(* PLC project prj, KAIST_DSLAB noNameNow 1, author bwkim *)
(* stored: creationDateTime 2015-7-21T04:57:08, modificationDateTime 2015-7-21T04:57:08 *)

PROGRAM program5____sub1
  VAR
    VF_TON : null;
  END_VAR
  VAR
    VF_PTON : null;
  END_VAR
  VAR_INPUT CONSTANT
    K_DELAY : null;
  END_VAR
  VAR_OUTPUT
    TON_et : null;
  END_VAR
  VAR_OUTPUT
    PTON_et : null;
  END_VAR
  VAR_IN_OUT
    PTRIP_LOGIC : BOOL := FALSE;
  END_VAR
  VAR_IN_OUT
    TRIP_LOGIC : BOOL := FALSE;
  END_VAR
  VAR  (* added by the conversion: wires and edge detectors of the diagram *)
    _SUB_REAL34_OUT : ANY;
    _DIV_REAL56_OUT : INT;
    _SEL_REAL72_OUT : INT;
    _SEL_REAL73_OUT : INT;
    _SEL_REAL74_OUT : INT;
    _SEL_BOOL75_OUT : BOOL;
    _SEL_REAL39_OUT : INT;
    _SEL_BOOL82_OUT : BOOL;
    _SEL_REAL83_OUT : INT;
    _AND2_BOOL63_OUT : BOOL;
    _SEL_REAL86_OUT : INT;
    _SEL_REAL87_OUT : INT;
    _AND2_BOOL41_OUT : ANY;
  END_VAR

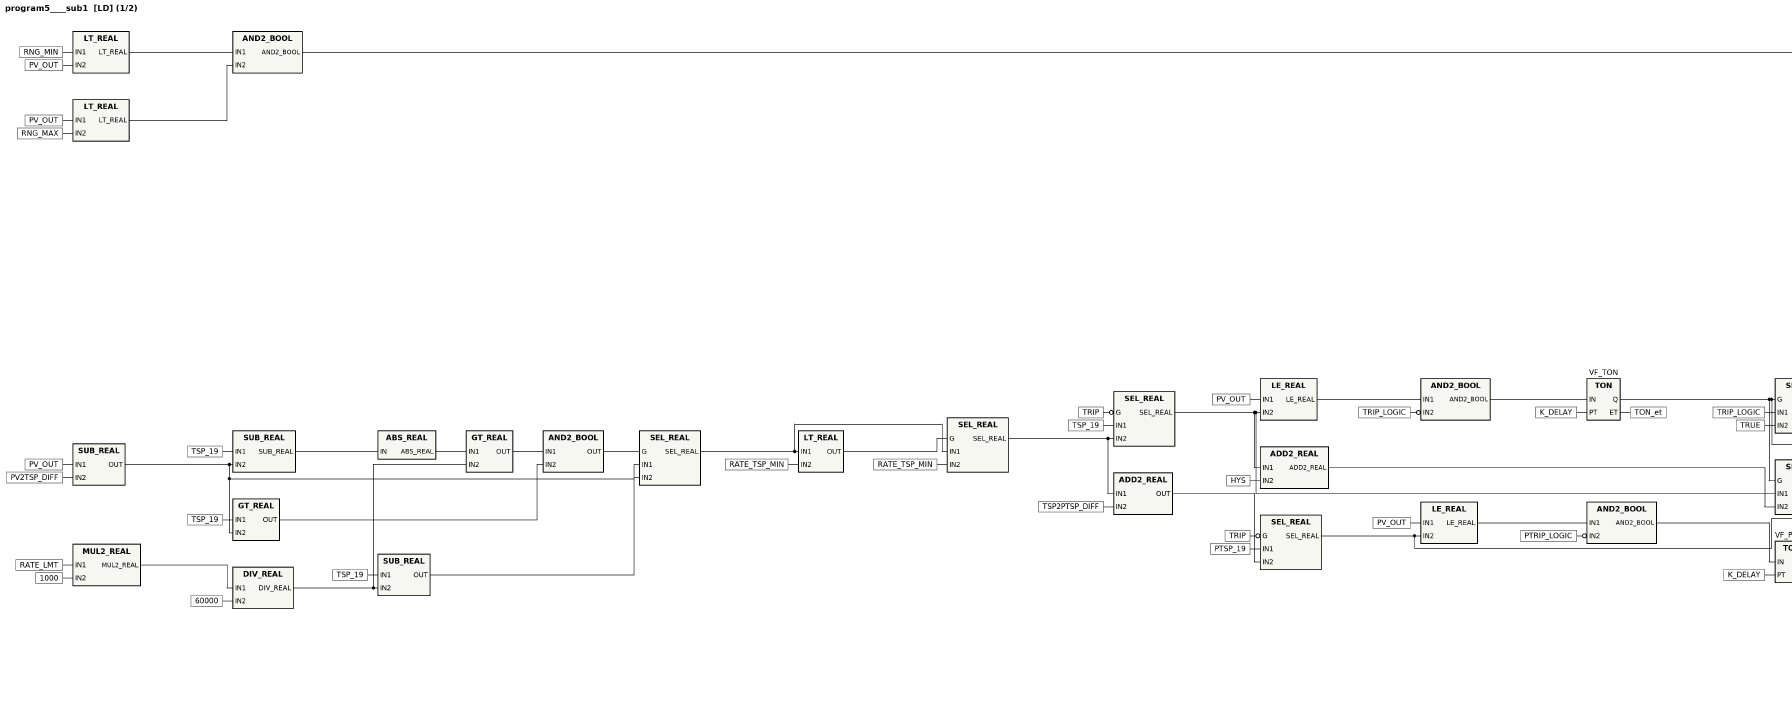
(* LD diagram, written out as Structured Text *)
_SUB_REAL34_OUT := SUB_REAL(PV_OUT, PV2TSP_DIFF);
_DIV_REAL56_OUT := DIV_REAL(MUL2_REAL(RATE_LMT, 1000), 60000);
_SEL_REAL72_OUT := SEL_REAL(AND2_BOOL(GT_REAL(ABS_REAL(SUB_REAL(TSP_19, _SUB_REAL34_OUT)), _DIV_REAL56_OUT), GT_REAL(TSP_19, _SUB_REAL34_OUT)), _SUB_REAL34_OUT, SUB_REAL(TSP_19, _DIV_REAL56_OUT));
_SEL_REAL73_OUT := SEL_REAL(LT_REAL(_SEL_REAL72_OUT, RATE_TSP_MIN), _SEL_REAL72_OUT, RATE_TSP_MIN);
_SEL_REAL74_OUT := SEL_REAL(NOT TRIP, PTSP_19, ADD2_REAL(_SEL_REAL73_OUT, TSP2PTSP_DIFF));
VF_PTON(IN := AND2_BOOL(LE_REAL(PV_OUT, _SEL_REAL74_OUT), NOT PTRIP_LOGIC), PT := K_DELAY);
_SEL_BOOL75_OUT := SEL_BOOL(VF_PTON.Q, PTRIP_LOGIC, TRUE);
PTRIP_LOGIC := _SEL_BOOL75_OUT;
PTON_et := VF_PTON.ET;
_SEL_REAL39_OUT := SEL_REAL(NOT TRIP, TSP_19, _SEL_REAL73_OUT);
VF_TON(IN := AND2_BOOL(LE_REAL(PV_OUT, _SEL_REAL39_OUT), NOT TRIP_LOGIC), PT := K_DELAY);
_SEL_BOOL82_OUT := SEL_BOOL(VF_TON.Q, TRIP_LOGIC, TRUE);
TRIP_LOGIC := _SEL_BOOL82_OUT;
TON_et := VF_TON.ET;
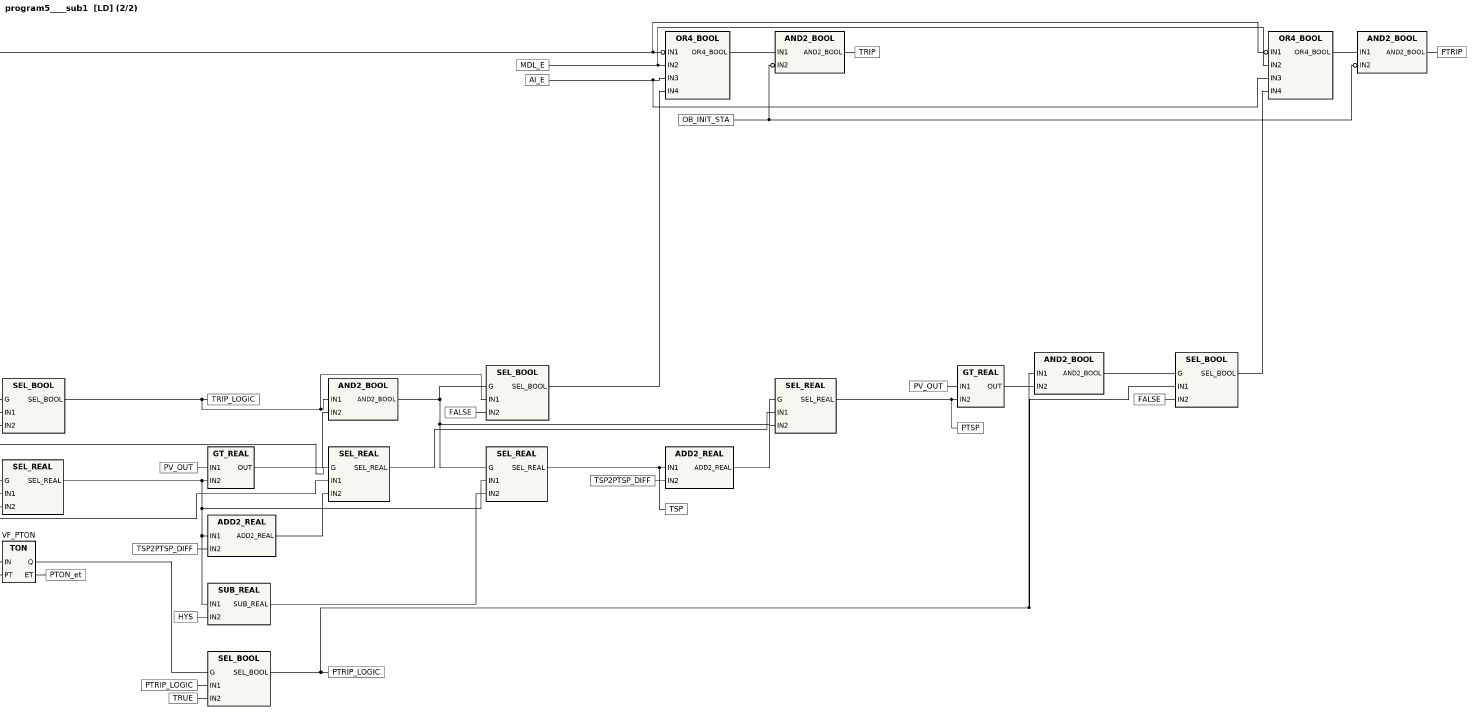
_SEL_REAL83_OUT := SEL_REAL(VF_TON.Q, _SEL_REAL39_OUT, ADD2_REAL(_SEL_REAL39_OUT, HYS));
_AND2_BOOL63_OUT := AND2_BOOL(_SEL_BOOL82_OUT, GT_REAL(PV_OUT, _SEL_REAL83_OUT));
_SEL_REAL86_OUT := SEL_REAL(_AND2_BOOL63_OUT, _SEL_REAL83_OUT, SUB_REAL(_SEL_REAL83_OUT, HYS));
TSP := _SEL_REAL86_OUT;
_SEL_REAL87_OUT := SEL_REAL(_AND2_BOOL63_OUT, SEL_REAL(VF_TON.Q, _SEL_REAL74_OUT, ADD2_REAL(_SEL_REAL83_OUT, TSP2PTSP_DIFF)), ADD2_REAL(_SEL_REAL86_OUT, TSP2PTSP_DIFF));
PTSP := _SEL_REAL87_OUT;
_AND2_BOOL41_OUT := AND2_BOOL(LT_REAL(RNG_MIN, PV_OUT), LT_REAL(PV_OUT, RNG_MAX));
PTRIP := AND2_BOOL(OR4_BOOL(NOT _AND2_BOOL41_OUT, MDL_E, AI_E, SEL_BOOL(AND2_BOOL(_SEL_BOOL75_OUT, GT_REAL(PV_OUT, _SEL_REAL87_OUT)), _SEL_BOOL75_OUT, FALSE)), NOT OB_INIT_STA);
TRIP := AND2_BOOL(OR4_BOOL(NOT _AND2_BOOL41_OUT, MDL_E, AI_E, SEL_BOOL(_AND2_BOOL63_OUT, _SEL_BOOL82_OUT, FALSE)), NOT OB_INIT_STA);
END_PROGRAM
